TYPE ST_TxHmiMru :
STRUCT
	status : DINT;
END_STRUCT
END_TYPE

(* stored: Version 1.1.0.1, ProductVersion 3.1.4022.7
   DUT ST_TxHmiMru: Id {d1813d09-0a0c-4b1f-98e8-7a953aea8dbc} *)
